FUNCTION FUN_ConvFourByteToReal32 : REAL
VAR_INPUT
	nValue1		:BYTE;				// Input Byte no 1
	nValue2		:BYTE;				// Input Byte no 2
	nValue3		:BYTE;				// Input Byte no 3
	nValue4		:BYTE;				// Input Byte no 4
END_VAR
VAR
	uData		:U_Convert_REAL32;	// Data variable used for conversion
END_VAR


// Save input bytes in data union
uData.arrByte[1] := nValue1;
uData.arrByte[2] := nValue2;
uData.arrByte[3] := nValue3;
uData.arrByte[4] := nValue4;

// Return value
FUN_ConvFourByteToReal32 := uData.fValue;

END_FUNCTION

(* stored: Version 1.1.0.1, ProductVersion 3.1.4024.12
   POU FUN_ConvFourByteToReal32: Id {148b1433-23b8-42e7-b885-36166ec42f38}, SpecialFunc None *)
